Yaskawa INFORM job: PARK.JBI

/JOB
//NAME PARK
//POS
///NPOS 1,0,0,0
///TOOL 0
///PULSE
C000=-625,25464,-5087,0,6563,1454
//INST
///DATE 2014/11/06 17:46
///ATTR 0,0,0,0,0,0,0,0,0,0,0,0,0,1,0,0
///FRAME BASE
NOP
*1
MOVJ C000 VJ=25.00 CONT
PAUSE
JUMP *1
END
